TYPE Basic_Input_typ : 	
	STRUCT 
		Command : Basic_Command_axis_typ;
		Parameter : Bacis_Parameter_axis_typ;
	END_STRUCT
END_TYPE

(* stored: Version 1.1.0.1, ProductVersion 3.1.4024.3
   DUT Basic_Input_typ: Id {552577bd-b0e4-0757-39d5-9cacefe606f8} *)
